AssertArrayResults.ReportResult(ExpectedsSize := DINT_TO_UDINT(SizeOfExpecteds),
                                ExpectedsTypeClass := IBaseLibrary.TypeClass.TYPE_ULINT,
                                ActualsSize := DINT_TO_UDINT(SizeOfActuals),
                                ActualsTypeClass := IBaseLibrary.TypeClass.TYPE_ULINT,
                                Message := Message,
                                TestInstancePath := TestInstancePath,
                                AlreadyReported => AlreadyReported);

IF NOT AlreadyReported AND NOT Equals THEN
    SetTestFailed(AssertionType := E_AssertionType.Type_Array_ULINT,
                  AssertionMessage := Message);

    IF NOT SizeEquals THEN
        Message := Tc2_Standard.CONCAT(STR1 := Message, STR2 := ', size of arrays not matching.');
        ExpectedString := 'SIZE = ';
        ExpectedString := Tc2_Standard.CONCAT(STR1 := ExpectedString, STR2 := DINT_TO_STRING(SizeOfExpecteds));
        ActualString := 'SIZE = ';
        ActualString := Tc2_Standard.CONCAT(STR1 := ActualString, STR2 := DINT_TO_STRING(SizeOfActuals));
    ELSE
        ExpectedString := 'ARRAY[';
        ExpectedString := Tc2_Standard.CONCAT(STR1 := ExpectedString, STR2 := DINT_TO_STRING(ExpectedsIndex));
        ExpectedString := Tc2_Standard.CONCAT(STR1 := ExpectedString, STR2 := '] = ');
        ExpectedString := Tc2_Standard.CONCAT(STR1 := ExpectedString, STR2 := ULINT_TO_STRING(Expecteds[ExpectedsIndex]));

        ActualString := 'ARRAY[';
        ActualString := Tc2_Standard.CONCAT(STR1 := ActualString, STR2 := DINT_TO_STRING(ActualsIndex));
        ActualString := Tc2_Standard.CONCAT(STR1 := ActualString, STR2 := '] = ');
        ActualString := Tc2_Standard.CONCAT(STR1 := ActualString, STR2 := ULINT_TO_STRING(Actuals[ActualsIndex]));
    END_IF

    AssertMessageFormatter.LogAssertFailure(Expected := ExpectedString,
                                            Actual := ActualString,
                                            Message := Message,
                                            TestInstancePath := TestInstancePath);
END_IF
END_METHOD

(*
    Asserts that two USINT arrays are equal. If they are not, an assertion error is created.
*)
METHOD PUBLIC AssertArrayEquals_USINT
VAR_IN_OUT
    Expecteds : ARRAY[*] OF USINT; // USINT array with expected values
    Actuals : ARRAY[*] OF USINT; // USINT array with actual values
END_VAR
VAR_INPUT
    Message : Tc2_System.T_MaxString; // The identifying message for the assertion error
END_VAR
VAR
    Equals : BOOL := TRUE;
    SizeEquals : BOOL := TRUE;
    Index : DINT;
    ExpectedString : Tc2_System.T_MaxString;
    ActualString : Tc2_System.T_MaxString;
    AlreadyReported : BOOL;
    TestInstancePath : Tc2_System.T_MaxString;
    SizeOfExpecteds : DINT;
    SizeOfActuals : DINT;
    ExpectedsIndex : DINT;
    ActualsIndex : DINT;
END_VAR
IF GVL_TcUnit.IgnoreCurrentTest OR GVL_TcUnit.CurrentTestIsFinished THEN
    RETURN;
END_IF

TestInstancePath := AddTestNameToInstancePath(FindTestSuiteInstancePath());

SizeOfExpecteds := ABS(UPPER_BOUND(Expecteds, 1) - LOWER_BOUND(Expecteds, 1)) + 1;
SizeOfActuals := ABS(UPPER_BOUND(Actuals, 1) - LOWER_BOUND(Actuals, 1)) + 1;

IF SizeOfExpecteds <> SizeOfActuals THEN
    Equals := FALSE;
    SizeEquals := FALSE;
ELSE
    (* Even though we know that both arrays are equal in size, the two arrays can start at two completely different
       indexes, which needs to be taken into account for. *)
    ExpectedsIndex := LOWER_BOUND(Expecteds, 1); // The start position for the expecteds
    ActualsIndex := LOWER_BOUND(Actuals, 1); // The start position for the actuals
    FOR Index := 1 TO SizeOfExpecteds BY 1 DO
        IF Expecteds[ExpectedsIndex] <> Actuals[ActualsIndex] THEN
            Equals := FALSE;
            EXIT;
        END_IF
        ExpectedsIndex := ExpectedsIndex + 1;
        ActualsIndex := ActualsIndex + 1;
    END_FOR
END_IF

AssertArrayResults.ReportResult(ExpectedsSize := DINT_TO_UDINT(SizeOfExpecteds),
                                ExpectedsTypeClass := IBaseLibrary.TypeClass.TYPE_USINT,
                                ActualsSize := DINT_TO_UDINT(SizeOfActuals),
                                ActualsTypeClass := IBaseLibrary.TypeClass.TYPE_USINT,
                                Message := Message,
                                TestInstancePath := TestInstancePath,
                                AlreadyReported => AlreadyReported);

IF NOT AlreadyReported AND NOT Equals THEN
    SetTestFailed(AssertionType := E_AssertionType.Type_Array_USINT,
                  AssertionMessage := Message);

    IF NOT SizeEquals THEN
        Message := Tc2_Standard.CONCAT(STR1 := Message, STR2 := ', size of arrays not matching.');
        ExpectedString := 'SIZE = ';
        ExpectedString := Tc2_Standard.CONCAT(STR1 := ExpectedString, STR2 := DINT_TO_STRING(SizeOfExpecteds));
        ActualString := 'SIZE = ';
        ActualString := Tc2_Standard.CONCAT(STR1 := ActualString, STR2 := DINT_TO_STRING(SizeOfActuals));
    ELSE
        ExpectedString := 'ARRAY[';
        ExpectedString := Tc2_Standard.CONCAT(STR1 := ExpectedString, STR2 := DINT_TO_STRING(ExpectedsIndex));
        ExpectedString := Tc2_Standard.CONCAT(STR1 := ExpectedString, STR2 := '] = ');
        ExpectedString := Tc2_Standard.CONCAT(STR1 := ExpectedString, STR2 := USINT_TO_STRING(Expecteds[ExpectedsIndex]));

        ActualString := 'ARRAY[';
        ActualString := Tc2_Standard.CONCAT(STR1 := ActualString, STR2 := DINT_TO_STRING(ActualsIndex));
        ActualString := Tc2_Standard.CONCAT(STR1 := ActualString, STR2 := '] = ');
        ActualString := Tc2_Standard.CONCAT(STR1 := ActualString, STR2 := USINT_TO_STRING(Actuals[ActualsIndex]));
    END_IF

    AssertMessageFormatter.LogAssertFailure(Expected := ExpectedString,
                                            Actual := ActualString,
                                            Message := Message,
                                            TestInstancePath := TestInstancePath);
END_IF
END_METHOD

(*
    Asserts that two WORD arrays are equal. If they are not, an assertion error is created.
*)
METHOD PUBLIC AssertArrayEquals_WORD
VAR_IN_OUT
    Expecteds : ARRAY[*] OF WORD; // WORD array with expected values
    Actuals : ARRAY[*] OF WORD; // WORD array with actual values
END_VAR
VAR_INPUT
    Message : Tc2_System.T_MaxString; // The identifying message for the assertion error
END_VAR
VAR
    Equals : BOOL := TRUE;
    SizeEquals : BOOL := TRUE;
    Index : DINT;
    ExpectedString : Tc2_System.T_MaxString;
    ActualString : Tc2_System.T_MaxString;
    AlreadyReported : BOOL;
    TestInstancePath : Tc2_System.T_MaxString;
    SizeOfExpecteds : DINT;
    SizeOfActuals : DINT;
    ExpectedDWordString : STRING;
    ActualDWordString : STRING;
    ExpectedsIndex : DINT;
    ActualsIndex : DINT;
END_VAR
IF GVL_TcUnit.IgnoreCurrentTest OR GVL_TcUnit.CurrentTestIsFinished THEN
    RETURN;
END_IF

TestInstancePath := AddTestNameToInstancePath(FindTestSuiteInstancePath());

SizeOfExpecteds := ABS(UPPER_BOUND(Expecteds, 1) - LOWER_BOUND(Expecteds, 1)) + 1;
SizeOfActuals := ABS(UPPER_BOUND(Actuals, 1) - LOWER_BOUND(Actuals, 1)) + 1;

IF SizeOfExpecteds <> SizeOfActuals THEN
    Equals := FALSE;
    SizeEquals := FALSE;
ELSE
    (* Even though we know that both arrays are equal in size, the two arrays can start at two completely different
       indexes, which needs to be taken into account for. *)
    ExpectedsIndex := LOWER_BOUND(Expecteds, 1); // The start position for the expecteds
    ActualsIndex := LOWER_BOUND(Actuals, 1); // The start position for the actuals
    FOR Index := 1 TO SizeOfExpecteds BY 1 DO
        IF Expecteds[ExpectedsIndex] <> Actuals[ActualsIndex] THEN
            Equals := FALSE;
            EXIT;
        END_IF
        ExpectedsIndex := ExpectedsIndex + 1;
        ActualsIndex := ActualsIndex + 1;
    END_FOR
END_IF

AssertArrayResults.ReportResult(ExpectedsSize := DINT_TO_UDINT(SizeOfExpecteds),
                                ExpectedsTypeClass := IBaseLibrary.TypeClass.TYPE_WORD,
                                ActualsSize := DINT_TO_UDINT(SizeOfActuals),
                                ActualsTypeClass := IBaseLibrary.TypeClass.TYPE_WORD,
                                Message := Message,
                                TestInstancePath := TestInstancePath,
                                AlreadyReported => AlreadyReported);

IF NOT AlreadyReported AND NOT Equals THEN
    SetTestFailed(AssertionType := E_AssertionType.Type_Array_WORD,
                  AssertionMessage := Message);

    IF NOT SizeEquals THEN
        Message := Tc2_System.CONCAT(STR1 := Message, STR2 := ', size of arrays not matching.');
        ExpectedString := 'SIZE = ';
        ExpectedString := Tc2_System.CONCAT(STR1 := ExpectedString, STR2 := DINT_TO_STRING(SizeOfExpecteds));
        ActualString := 'SIZE = ';
        ActualString := Tc2_System.CONCAT(STR1 := ActualString, STR2 := DINT_TO_STRING(SizeOfActuals));
    ELSE
        ExpectedDWordString := Tc2_Standard.CONCAT(STR1 := '0x',
                                                  STR2 := Tc2_Utilities.WORD_TO_HEXSTR(in := Expecteds[ExpectedsIndex],
                                                                                       iPrecision := 4,
                                                                                       bLoCase := FALSE));
        ExpectedString := 'ARRAY[';
        ExpectedString := Tc2_System.CONCAT(STR1 := ExpectedString, STR2 := DINT_TO_STRING(ExpectedsIndex));
        ExpectedString := Tc2_System.CONCAT(STR1 := ExpectedString, STR2 := '] = ');
        ExpectedString := Tc2_System.CONCAT(STR1 := ExpectedString, STR2 := ExpectedDWordString);

        ActualDWordString := Tc2_Standard.CONCAT(STR1 := '0x',
                                                 STR2 := Tc2_Utilities.WORD_TO_HEXSTR(in := Actuals[ActualsIndex],
                                                                                      iPrecision := 4,
                                                                                      bLoCase := FALSE));
        ActualString := 'ARRAY[';
        ActualString := Tc2_System.CONCAT(STR1 := ActualString, STR2 := DINT_TO_STRING(ActualsIndex));
        ActualString := Tc2_System.CONCAT(STR1 := ActualString, STR2 := '] = ');
        ActualString := Tc2_System.CONCAT(STR1 := ActualString, STR2 := ActualDWordString);
    END_IF

    AssertMessageFormatter.LogAssertFailure(Expected := ExpectedString,
                                            Actual := ActualString,
                                            Message := Message,
                                            TestInstancePath := TestInstancePath);
END_IF
END_METHOD

(*
    Asserts that two objects (of any type) are equal. If they are not, an assertion error is created.
    For REAL and LREAL it's recommended to use the AssertEquals_REAL or AssertEquals_LREAL respectively
    as these give the possibility to specify a delta between the expected and actual value.
*)
METHOD PUBLIC AssertEquals
VAR_INPUT
    Expected : ANY; // Expected value
    Actual : ANY; // The value to check against expected
    Message : Tc2_System.T_MaxString; // The identifying message for the assertion error
END_VAR
VAR
    Count : DINT;
    ExpectedDataString : Tc2_System.T_MaxString;
    ActualDataString : Tc2_System.T_MaxString;
    TestInstancePath : Tc2_System.T_MaxString;
    AlreadyReported : BOOL;

    boolExpected : BOOL;
    boolActual : BOOL;
    byteExpected : BYTE;
    byteActual : BYTE;
    dateExpected : DATE;
    dateActual : DATE;
    dateAndTimeExpected : DATE_AND_TIME;
    dateAndTimeActual : DATE_AND_TIME;
    dintExpected : DINT;
    dintActual : DINT;
    dwordExpected : DWORD;
    dwordActual : DWORD;
    intExpected : INT;
    intActual : INT;
    lintExpected : LINT;
    lintActual : LINT;
    lrealExpected : LREAL;
    lrealActual : LREAL;
    ltimeExpected : LTIME;
    ltimeActual : LTIME;
    lwordExpected : LWORD;
    lwordActual : LWORD;
    realExpected : REAL;
    realActual : REAL;
    sintExpected : SINT;
    sintActual : SINT;
    stringExpected : Tc2_System.T_MaxString;
    stringActual : Tc2_System.T_MaxString;
    wstringExpected : WSTRING(255);
    wstringActual : WSTRING(255);
    timeExpected : TIME;
    timeActual : TIME;
    timeOfDayExpected : TIME_OF_DAY;
    timeOfDayActual : TIME_OF_DAY;
    udintExpected : UDINT;
    udintActual : UDINT;
    uintExpected : UINT;
    uintActual : UINT;
    ulintExpected : ULINT;
    ulintActual : ULINT;
    usintExpected : USINT;
    usintActual : USINT;
    wordExpected : WORD;
    wordActual : WORD;

    (* ANY comparison variables *)
    DataTypesNotEquals : BOOL; // The data type of the two ANY input parameters are not equal
    DataSizeNotEquals : BOOL; // The data size of the two ANY input parameters are not equal
    DataContentNotEquals : BOOL; // The data content of the two ANY input parameters are not equal
    IteratorCounter : DINT;
END_VAR
IF GVL_TcUnit.IgnoreCurrentTest OR GVL_TcUnit.CurrentTestIsFinished THEN
    RETURN;
END_IF

(*
    This compares two instances of any object type and returns whether they
    are the same type, size and value or not. This is necessary for two reasons:
    1. So that we can know exactly what differs between the two input parameters
    2. It's not possible to do a comparison (= or <>) between two instances of ANY. 
*)
(* Check whether the type of the inputs differs *)
IF Expected.TypeClass <> Actual.TypeClass THEN
    DataTypesNotEquals := TRUE;
END_IF

(* Check whether the size of the inputs differs *)
IF NOT DataTypesNotEquals THEN
    (* Take special care of STRING and WSTRING, as these can be declared with different sizes,
       although their content might be the same *)
    IF UDINT_TO_INT(Expected.TypeClass) = IBaseLibrary.TypeClass.TYPE_STRING THEN
        Tc2_System.MEMCPY(destAddr := ADR(stringExpected), srcAddr := Expected.pValue, n := DINT_TO_UDINT(Expected.diSize));
        Tc2_System.MEMCPY(destAddr := ADR(stringActual), srcAddr := Actual.pValue, n := DINT_TO_UDINT(Actual.diSize));
        DataSizeNotEquals := Tc2_Standard.LEN(STR := stringExpected) <> Tc2_Standard.LEN(STR := stringActual);
    ELSIF UDINT_TO_INT(Expected.TypeClass) = IBaseLibrary.TypeClass.TYPE_WSTRING THEN
        Tc2_System.MEMCPY(destAddr := ADR(wstringExpected), srcAddr := Expected.pValue, n := DINT_TO_UDINT(Expected.diSize));
        Tc2_System.MEMCPY(destAddr := ADR(wstringActual), srcAddr := Actual.pValue, n := DINT_TO_UDINT(Actual.diSize));
        DataSizeNotEquals := Tc2_Standard.WLEN(STR := wstringExpected) <> Tc2_Standard.WLEN(STR := wstringActual);
    ELSIF (Expected.diSize <> Actual.diSize) THEN
        DataSizeNotEquals := TRUE;
    END_IF
END_IF

(* Even though the data type and size are equals, the contents may still differ *)
IF NOT DataTypesNotEquals AND NOT DataSizeNotEquals THEN
    // Compare each byte in the ANY-types
    FOR IteratorCounter := 0 TO Expected.diSize - 1 BY 1 DO
        IF Expected.pValue[IteratorCounter] <> Actual.pValue[IteratorCounter] THEN
            DataContentNotEquals := TRUE;
            EXIT;
        END_IF
    END_FOR
END_IF

(* First check whether the input data are any of the standard data types that are supported by TcUnit.
   In this case call the standard Assert-methods for that data. But before doing that we need to make sure
   that both the expected and actual:
   - Have both the same data type
   - Both have the same data size
*)
IF NOT DataTypesNotEquals AND NOT DataSizeNotEquals THEN

    (* BOOL *)
    IF UDINT_TO_INT(Expected.TypeClass) = IBaseLibrary.TypeClass.TYPE_BOOL THEN
        Tc2_System.MEMCPY(destAddr := ADR(boolExpected), srcAddr := Expected.pValue, n := SIZEOF(BOOL));
        Tc2_System.MEMCPY(destAddr := ADR(boolActual), srcAddr := Actual.pValue, n := SIZEOF(BOOL));
        AssertEquals_BOOL(Expected := boolExpected, Actual := boolActual, Message := Message);
        RETURN;
    END_IF

    (* BYTE *)
    IF UDINT_TO_INT(Expected.TypeClass) = IBaseLibrary.TypeClass.TYPE_BYTE THEN
        Tc2_System.MEMCPY(destAddr := ADR(byteExpected), srcAddr := Expected.pValue, n := SIZEOF(BYTE));
        Tc2_System.MEMCPY(destAddr := ADR(byteActual), srcAddr := Actual.pValue, n := SIZEOF(BYTE));
        AssertEquals_BYTE(Expected := byteExpected, Actual := byteActual, Message := Message);
        RETURN;
    END_IF

    (* DATE *)
    IF UDINT_TO_INT(Expected.TypeClass) = IBaseLibrary.TypeClass.TYPE_DATE THEN
        Tc2_System.MEMCPY(destAddr := ADR(dateExpected), srcAddr := Expected.pValue, n := SIZEOF(DATE));
        Tc2_System.MEMCPY(destAddr := ADR(dateActual), srcAddr := Actual.pValue, n := SIZEOF(DATE));
        AssertEquals_DATE(Expected := dateExpected, Actual := dateActual, Message := Message);
        RETURN;
    END_IF

    (* DATE_AND_TIME *)
    IF UDINT_TO_INT(Expected.TypeClass) = IBaseLibrary.TypeClass.TYPE_DATEANDTIME THEN
        Tc2_System.MEMCPY(destAddr := ADR(dateAndTimeExpected), srcAddr := Expected.pValue, n := SIZEOF(DATE_AND_TIME));
        Tc2_System.MEMCPY(destAddr := ADR(dateAndTimeActual), srcAddr := Actual.pValue, n := SIZEOF(DATE_AND_TIME));
        AssertEquals_DATE_AND_TIME(Expected := dateAndTimeExpected, Actual := dateAndTimeActual, Message := Message);
        RETURN;
    END_IF

    (* DINT *)
    IF UDINT_TO_INT(Expected.TypeClass) = IBaseLibrary.TypeClass.TYPE_DINT THEN
        Tc2_System.MEMCPY(destAddr := ADR(dintExpected), srcAddr := Expected.pValue, n := SIZEOF(DINT));
        Tc2_System.MEMCPY(destAddr := ADR(dintActual), srcAddr := Actual.pValue, n := SIZEOF(DINT));
        AssertEquals_DINT(Expected := dintExpected, Actual := dintActual, Message := Message);
        RETURN;
    END_IF

    (* DWORD *)
    IF UDINT_TO_INT(Expected.TypeClass) = IBaseLibrary.TypeClass.TYPE_DWORD THEN
        Tc2_System.MEMCPY(destAddr := ADR(dwordExpected), srcAddr := Expected.pValue, n := SIZEOF(DWORD));
        Tc2_System.MEMCPY(destAddr := ADR(dwordActual), srcAddr := Actual.pValue, n := SIZEOF(DWORD));
        AssertEquals_DWORD(Expected := dwordExpected, Actual := dwordActual, Message := Message);
        RETURN;
    END_IF

    (* INT *)
    IF UDINT_TO_INT(Expected.TypeClass) = IBaseLibrary.TypeClass.TYPE_INT THEN
        Tc2_System.MEMCPY(destAddr := ADR(intExpected), srcAddr := Expected.pValue, n := SIZEOF(INT));
        Tc2_System.MEMCPY(destAddr := ADR(intActual), srcAddr := Actual.pValue, n := SIZEOF(INT));
        AssertEquals_INT(Expected := intExpected, Actual := intActual, Message := Message);
        RETURN;
    END_IF

    (* LINT *)
    IF UDINT_TO_INT(Expected.TypeClass) = IBaseLibrary.TypeClass.TYPE_LINT THEN
        Tc2_System.MEMCPY(destAddr := ADR(lintExpected), srcAddr := Expected.pValue, n := SIZEOF(LINT));
        Tc2_System.MEMCPY(destAddr := ADR(lintActual), srcAddr := Actual.pValue, n := SIZEOF(LINT));
        AssertEquals_LINT(Expected := lintExpected, Actual := lintActual, Message := Message);
        RETURN;
    END_IF

    (* LREAL *)
    IF UDINT_TO_INT(Expected.TypeClass) = IBaseLibrary.TypeClass.TYPE_LREAL THEN
        Tc2_System.MEMCPY(destAddr := ADR(lrealExpected), srcAddr := Expected.pValue, n := SIZEOF(LREAL));
        Tc2_System.MEMCPY(destAddr := ADR(lrealActual), srcAddr := Actual.pValue, n := SIZEOF(LREAL));
        AssertEquals_LREAL(Expected := lrealExpected, Actual := lrealActual, Delta := 0.0, Message := Message);
        RETURN;
    END_IF

    (* LTIME *)
    IF UDINT_TO_INT(Expected.TypeClass) = IBaseLibrary.TypeClass.TYPE_LTIME THEN
        Tc2_System.MEMCPY(destAddr := ADR(ltimeExpected), srcAddr := Expected.pValue, n := SIZEOF(LTIME));
        Tc2_System.MEMCPY(destAddr := ADR(ltimeActual), srcAddr := Actual.pValue, n := SIZEOF(LTIME));
        AssertEquals_LTIME(Expected := ltimeExpected, Actual := ltimeActual, Message := Message);
        RETURN;
    END_IF

    (* LWORD *)
    IF UDINT_TO_INT(Expected.TypeClass) = IBaseLibrary.TypeClass.TYPE_LWORD THEN
        Tc2_System.MEMCPY(destAddr := ADR(lwordExpected), srcAddr := Expected.pValue, n := SIZEOF(LWORD));
        Tc2_System.MEMCPY(destAddr := ADR(lwordActual), srcAddr := Actual.pValue, n := SIZEOF(LWORD));
        AssertEquals_LWORD(Expected := lwordExpected, Actual := lwordActual, Message := Message);
        RETURN;
    END_IF

    (* REAL *)
    IF UDINT_TO_INT(Expected.TypeClass) = IBaseLibrary.TypeClass.TYPE_REAL THEN
        Tc2_System.MEMCPY(destAddr := ADR(realExpected), srcAddr := Expected.pValue, n := SIZEOF(REAL));
        Tc2_System.MEMCPY(destAddr := ADR(realActual), srcAddr := Actual.pValue, n := SIZEOF(REAL));
        AssertEquals_REAL(Expected := realExpected, Actual := realActual, Delta := 0.0, Message := Message);
        RETURN;
    END_IF

    (* SINT *)
    IF UDINT_TO_INT(Expected.TypeClass) = IBaseLibrary.TypeClass.TYPE_SINT THEN
        Tc2_System.MEMCPY(destAddr := ADR(sintExpected), srcAddr := Expected.pValue, n := SIZEOF(SINT));
        Tc2_System.MEMCPY(destAddr := ADR(sintActual), srcAddr := Actual.pValue, n := SIZEOF(SINT));
        AssertEquals_SINT(Expected := sintExpected, Actual := sintActual, Message := Message);
        RETURN;
    END_IF

    (* STRING *)
    IF UDINT_TO_INT(Expected.TypeClass) = IBaseLibrary.TypeClass.TYPE_STRING THEN
        Tc2_System.MEMCPY(destAddr := ADR(stringExpected), srcAddr := Expected.pValue, n := DINT_TO_UDINT(Expected.diSize));
        Tc2_System.MEMCPY(destAddr := ADR(stringActual), srcAddr := Actual.pValue, n := DINT_TO_UDINT(Actual.diSize));
        AssertEquals_STRING(Expected := stringExpected, Actual := stringActual, Message := Message);
        RETURN;
    END_IF

    (* WSTRING *)
    IF UDINT_TO_INT(Expected.TypeClass) = IBaseLibrary.TypeClass.TYPE_WSTRING THEN
        Tc2_System.MEMCPY(destAddr := ADR(wstringExpected), srcAddr := Expected.pValue, n := DINT_TO_UDINT(Expected.diSize));
        Tc2_System.MEMCPY(destAddr := ADR(wstringActual), srcAddr := Actual.pValue, n := DINT_TO_UDINT(Actual.diSize));
        AssertEquals_WSTRING(Expected := wstringExpected, Actual := wstringActual, Message := Message);
        RETURN;
    END_IF

    (* TIME *)
    IF UDINT_TO_INT(Expected.TypeClass) = IBaseLibrary.TypeClass.TYPE_TIME THEN
        Tc2_System.MEMCPY(destAddr := ADR(timeExpected), srcAddr := Expected.pValue, n := SIZEOF(TIME));
        Tc2_System.MEMCPY(destAddr := ADR(timeActual), srcAddr := Actual.pValue, n := SIZEOF(TIME));
        AssertEquals_TIME(Expected := timeExpected, Actual := timeActual, Message := Message);
        RETURN;
    END_IF

    (* TIME_OF_DAY *)
    IF UDINT_TO_INT(Expected.TypeClass) = IBaseLibrary.TypeClass.TYPE_TIMEOFDAY THEN
        Tc2_System.MEMCPY(destAddr := ADR(timeOfDayExpected), srcAddr := Expected.pValue, n := SIZEOF(TIME_OF_DAY));
        Tc2_System.MEMCPY(destAddr := ADR(timeOfDayActual), srcAddr := Actual.pValue, n := SIZEOF(TIME_OF_DAY));
        AssertEquals_TIME_OF_DAY(Expected := timeOfDayExpected, Actual := timeOfDayActual, Message := Message);
        RETURN;
    END_IF

    (* UDINT *)
    IF UDINT_TO_INT(Expected.TypeClass) = IBaseLibrary.TypeClass.TYPE_UDINT THEN
        Tc2_System.MEMCPY(destAddr := ADR(udintExpected), srcAddr := Expected.pValue, n := SIZEOF(UDINT));
        Tc2_System.MEMCPY(destAddr := ADR(udintActual), srcAddr := Actual.pValue, n := SIZEOF(UDINT));
        AssertEquals_UDINT(Expected := udintExpected, Actual := udintActual, Message := Message);
        RETURN;
    END_IF

    (* UINT *)
    IF UDINT_TO_INT(Expected.TypeClass) = IBaseLibrary.TypeClass.TYPE_UINT THEN
        Tc2_System.MEMCPY(destAddr := ADR(uintExpected), srcAddr := Expected.pValue, n := SIZEOF(UINT));
        Tc2_System.MEMCPY(destAddr := ADR(uintActual), srcAddr := Actual.pValue, n := SIZEOF(UINT));
        AssertEquals_UINT(Expected := uintExpected, Actual := uintActual, Message := Message);
        RETURN;
    END_IF

    (* ULINT *)
    IF UDINT_TO_INT(Expected.TypeClass) = IBaseLibrary.TypeClass.TYPE_ULINT THEN
        Tc2_System.MEMCPY(destAddr := ADR(ulintExpected), srcAddr := Expected.pValue, n := SIZEOF(ULINT));
        Tc2_System.MEMCPY(destAddr := ADR(ulintActual), srcAddr := Actual.pValue, n := SIZEOF(ULINT));
        AssertEquals_ULINT(Expected := ulintExpected, Actual := ulintActual, Message := Message);
        RETURN;
    END_IF

    (* USINT *)
    IF UDINT_TO_INT(Expected.TypeClass) = IBaseLibrary.TypeClass.TYPE_USINT THEN
        Tc2_System.MEMCPY(destAddr := ADR(usintExpected), srcAddr := Expected.pValue, n := SIZEOF(USINT));
        Tc2_System.MEMCPY(destAddr := ADR(usintActual), srcAddr := Actual.pValue, n := SIZEOF(USINT));
        AssertEquals_USINT(Expected := usintExpected, Actual := usintActual, Message := Message);
        RETURN;
    END_IF

    (* WORD *)
    IF UDINT_TO_INT(Expected.TypeClass) = IBaseLibrary.TypeClass.TYPE_WORD THEN
        Tc2_System.MEMCPY(destAddr := ADR(wordExpected), srcAddr := Expected.pValue, n := SIZEOF(WORD));
        Tc2_System.MEMCPY(destAddr := ADR(wordActual), srcAddr := Actual.pValue, n := SIZEOF(WORD));
        AssertEquals_WORD(Expected := wordExpected, Actual := wordActual, Message := Message);
        RETURN;
    END_IF

END_IF

(* If we've come to this row, it means that the data input is not any of the standard primitive data types, and thus
   we need to do special handling *)
TestInstancePath := AddTestNameToInstancePath(TestInstancePath := FindTestSuiteInstancePath());

IF DataTypesNotEquals THEN
    ExpectedDataString := Tc2_Standard.CONCAT(STR1 := '(Type class = ', STR2 := F_AnyTypeClassToString((Expected.TypeClass)));
    ExpectedDataString := Tc2_Standard.CONCAT(STR1 := ExpectedDataString, STR2 := ')');
    ActualDataString := Tc2_Standard.CONCAT(STR1 := '(Type class = ', STR2 := F_AnyTypeClassToString(Actual.TypeClass));
    ActualDataString := Tc2_Standard.CONCAT(STR1 := ActualDataString, STR2 := ')');
ELSIF DataSizeNotEquals THEN
    (* Take special care of STRING and WSTRING, as these can be declared with different sizes,
       although their content might be the same *)
    IF UDINT_TO_INT(Expected.TypeClass) = IBaseLibrary.TypeClass.TYPE_STRING THEN
        Tc2_System.MEMCPY(destAddr := ADR(stringExpected), srcAddr := Expected.pValue, n := DINT_TO_UDINT(Expected.diSize));
        Tc2_System.MEMCPY(destAddr := ADR(stringActual), srcAddr := Actual.pValue, n := DINT_TO_UDINT(Actual.diSize));
        ExpectedDataString := Tc2_Standard.CONCAT(STR1 := '(Data size (LEN) = ', STR2 := INT_TO_STRING(Tc2_Standard.LEN(STR := stringExpected)));
        ActualDataString := Tc2_Standard.CONCAT(STR1 := '(Data size (LEN) = ', STR2 := INT_TO_STRING(Tc2_Standard.LEN(STR := stringActual)));
    ELSIF UDINT_TO_INT(Expected.TypeClass) = IBaseLibrary.TypeClass.TYPE_WSTRING THEN
        Tc2_System.MEMCPY(destAddr := ADR(wstringExpected), srcAddr := Expected.pValue, n := DINT_TO_UDINT(Expected.diSize));
        Tc2_System.MEMCPY(destAddr := ADR(wstringActual), srcAddr := Actual.pValue, n := DINT_TO_UDINT(Actual.diSize));
        ExpectedDataString := Tc2_Standard.CONCAT(STR1 := '(Data size (WLEN) = ', STR2 := INT_TO_STRING(Tc2_Standard.WLEN(STR := wstringExpected)));
        ActualDataString := Tc2_Standard.CONCAT(STR1 := '(Data size (WLEN) = ', STR2 := INT_TO_STRING(Tc2_Standard.WLEN(STR := wstringActual)));
    ELSE
        ExpectedDataString := Tc2_Standard.CONCAT(STR1 := '(Data size = ', STR2 := DINT_TO_STRING(Expected.diSize));
        ActualDataString := Tc2_Standard.CONCAT(STR1 := '(Data size = ', STR2 := DINT_TO_STRING(Actual.diSize));
    END_IF
    ExpectedDataString := Tc2_Standard.CONCAT(STR1 := ExpectedDataString, STR2 := ')');
    ActualDataString := Tc2_Standard.CONCAT(STR1 := ActualDataString, STR2 := ')');
ELSIF DataContentNotEquals THEN
    FOR Count := 0 TO MIN(Expected.diSize-1, 38) BY 1 DO // One byte will equal two characters (example: 255 = 0xff, 1 = 0x01)
        ExpectedDataString := Tc2_Standard.CONCAT(STR1 := ExpectedDataString,
                                                  STR2 := Tc2_Utilities.BYTE_TO_HEXSTR(in := Expected.pValue[Count],
                                                                                       iPrecision := 2,
                                                                                       bLoCase := FALSE));
    END_FOR
    ExpectedDataString := Tc2_Standard.CONCAT(STR1 := '0x', STR2 := ExpectedDataString);

    FOR Count := 0 TO MIN(Actual.diSize-1, 38) BY 1 DO // One byte will equal two characters (example: 255 = 0xff, 1 = 0x01)
        ActualDataString := Tc2_Standard.CONCAT(STR1 := ActualDataString,
                                                STR2 := Tc2_Utilities.BYTE_TO_HEXSTR(in := Actual.pValue[Count],
                                                                                     iPrecision := 2,
                                                                                     bLoCase := FALSE));
    END_FOR
    ActualDataString := Tc2_Standard.CONCAT(STR1 := '0x', STR2 := ActualDataString);
END_IF

AssertResults.ReportResult(ExpectedSize := DINT_TO_UDINT(Expected.diSize),
                           ExpectedTypeClass := UDINT_TO_INT(Expected.TypeClass),
                           ExpectedValue := Expected.pValue,
                           ActualSize := DINT_TO_UDINT(Actual.diSize),
                           ActualTypeClass := UDINT_TO_INT(Actual.TypeClass),
                           ActualValue := Actual.pValue,
                           Message := Message,
                           TestInstancePath := TestInstancePath,
                           AlreadyReported => AlreadyReported);

IF NOT AlreadyReported AND (DataTypesNotEquals OR DataSizeNotEquals OR DataContentNotEquals) THEN
    SetTestFailed(AssertionType := E_AssertionType.Type_ANY,
                  AssertionMessage := Message);

    AssertMessageFormatter.LogAssertFailure(Expected := ExpectedDataString,
                                            Actual := ActualDataString,
                                            Message := Message,
                                            TestInstancePath := TestInstancePath);
END_IF
END_METHOD

(*
    Asserts that two BOOLs are equal. If they are not, an assertion error is created.
*)
METHOD PUBLIC AssertEquals_BOOL
VAR_INPUT
    Expected : BOOL; // BOOL expected value
    Actual : BOOL; // BOOL actual value
    Message : Tc2_System.T_MaxString; // The identifying message for the assertion error
END_VAR
VAR
    AlreadyReported : BOOL;
    TestInstancePath : Tc2_System.T_MaxString;
END_VAR
IF GVL_TcUnit.IgnoreCurrentTest OR GVL_TcUnit.CurrentTestIsFinished THEN
    RETURN;
END_IF

TestInstancePath := AddTestNameToInstancePath(TestInstancePath := FindTestSuiteInstancePath());

AssertResults.ReportResult(ExpectedSize := SIZEOF(Expected),
                           ExpectedTypeClass := IBaseLibrary.TypeClass.TYPE_BOOL,
                           ExpectedValue := ADR(Expected),
                           ActualSize := SIZEOF(Actual),
                           ActualTypeClass := IBaseLibrary.TypeClass.TYPE_BOOL,
                           ActualValue := ADR(Actual),
                           Message := Message,
                           TestInstancePath := TestInstancePath,
                           AlreadyReported => AlreadyReported);

IF NOT AlreadyReported AND Expected <> Actual THEN
    SetTestFailed(AssertionType := E_AssertionType.Type_BOOL,
                  AssertionMessage := Message);

    AssertMessageFormatter.LogAssertFailure(Expected := BOOL_TO_STRING(Expected),
                                            Actual := BOOL_TO_STRING(Actual),
                                            Message := Message,
                                            TestInstancePath := TestInstancePath);
END_IF
END_METHOD

(*
    Asserts that two BYTEs are equal. If they are not, an assertion error is created.
*)
METHOD PUBLIC AssertEquals_BYTE
VAR_INPUT
    Expected : BYTE; // BYTE expected value
    Actual : BYTE; // BYTE actual value
    Message : Tc2_System.T_MaxString; // The identifying message for the assertion error
END_VAR
VAR
    TestInstancePath : Tc2_System.T_MaxString;
    AlreadyReported : BOOL;
END_VAR
IF GVL_TcUnit.IgnoreCurrentTest OR GVL_TcUnit.CurrentTestIsFinished THEN
    RETURN;
END_IF

TestInstancePath := AddTestNameToInstancePath(TestInstancePath := FindTestSuiteInstancePath());

AssertResults.ReportResult(ExpectedSize := SIZEOF(Expected),
                           ExpectedTypeClass := IBaseLibrary.TypeClass.TYPE_BYTE,
                           ExpectedValue := ADR(Expected),
                           ActualSize := SIZEOF(Actual),
                           ActualTypeClass := IBaseLibrary.TypeClass.TYPE_BYTE,
                           ActualValue := ADR(Actual),
                           Message := Message,
                           TestInstancePath := TestInstancePath,
                           AlreadyReported => AlreadyReported);

IF NOT AlreadyReported AND Expected <> Actual THEN
    SetTestFailed(AssertionType := E_AssertionType.Type_BYTE,
                  AssertionMessage := Message);

    AssertMessageFormatter.LogAssertFailure(Expected := Tc2_Standard.CONCAT(
                                                       STR1 := '0x',
                                                       STR2 := Tc2_Utilities.BYTE_TO_HEXSTR(in := Expected,
                                                                                            iPrecision := 2,
                                                                                            bLoCase := FALSE)),
                                            Actual := Tc2_Standard.CONCAT(
                                                       STR1 := '0x',
                                                       STR2 := Tc2_Utilities.BYTE_TO_HEXSTR(in := Actual,
                                                                                            iPrecision := 2,
                                                                                            bLoCase := FALSE)),
                                            Message := Message,
                                            TestInstancePath := TestInstancePath);
END_IF
END_METHOD

(*
    Asserts that two DATEs are equal. If they are not, an assertion error is created.
*)
METHOD PUBLIC AssertEquals_DATE
VAR_INPUT
    Expected : DATE; // DATE expected value
    Actual : DATE; // DATE actual value
    Message : Tc2_System.T_MaxString; // The identifying message for the assertion error
END_VAR
VAR
    TestInstancePath : Tc2_System.T_MaxString;
    AlreadyReported : BOOL;
END_VAR
IF GVL_TcUnit.IgnoreCurrentTest OR GVL_TcUnit.CurrentTestIsFinished THEN
    RETURN;
END_IF

TestInstancePath := AddTestNameToInstancePath(TestInstancePath := FindTestSuiteInstancePath());

AssertResults.ReportResult(ExpectedSize := SIZEOF(Expected),
                           ExpectedTypeClass := IBaseLibrary.TypeClass.TYPE_DATE,
                           ExpectedValue := ADR(Expected),
                           ActualSize := SIZEOF(Actual),
                           ActualTypeClass := IBaseLibrary.TypeClass.TYPE_DATE,
                           ActualValue := ADR(Actual),
                           Message := Message,
                           TestInstancePath := TestInstancePath,
                           AlreadyReported => AlreadyReported);

IF NOT AlreadyReported AND Expected <> Actual THEN
    SetTestFailed(AssertionType := E_AssertionType.Type_DATE,
                  AssertionMessage := Message);

    AssertMessageFormatter.LogAssertFailure(Expected := DATE_TO_STRING(Expected),
                                            Actual := DATE_TO_STRING(Actual),
                                            Message := Message,
                                            TestInstancePath := TestInstancePath);
END_IF
END_METHOD

(*
    Asserts that two DATE_AND_TIMEs are equal. If they are not, an assertion error is created.
*)
METHOD PUBLIC AssertEquals_DATE_AND_TIME
VAR_INPUT
    Expected : DATE_AND_TIME; // DATE_AND_TIME expected value
    Actual : DATE_AND_TIME; // DATE_AND_TIME actual value
    Message : Tc2_System.T_MaxString; // The identifying message for the assertion error
END_VAR
VAR
    TestInstancePath : Tc2_System.T_MaxString;
    AlreadyReported : BOOL;
END_VAR
IF GVL_TcUnit.IgnoreCurrentTest OR GVL_TcUnit.CurrentTestIsFinished THEN
    RETURN;
END_IF

TestInstancePath := AddTestNameToInstancePath(TestInstancePath := FindTestSuiteInstancePath());

AssertResults.ReportResult(ExpectedSize := SIZEOF(Expected),
                           ExpectedTypeClass := IBaseLibrary.TypeClass.TYPE_DATEANDTIME,
                           ExpectedValue := ADR(Expected),
                           ActualSize := SIZEOF(Actual),
                           ActualTypeClass := IBaseLibrary.TypeClass.TYPE_DATEANDTIME,
                           ActualValue := ADR(Actual),
                           Message := Message,
                           TestInstancePath := TestInstancePath,
                           AlreadyReported => AlreadyReported);

IF NOT AlreadyReported AND Expected <> Actual THEN
    SetTestFailed(AssertionType := E_AssertionType.Type_DATE_AND_TIME,
                  AssertionMessage := Message);

    AssertMessageFormatter.LogAssertFailure(Expected := DT_TO_STRING(Expected),
                                            Actual := DT_TO_STRING(Actual),
                                            Message := Message,
                                            TestInstancePath := TestInstancePath);
END_IF
END_METHOD

(*
    Asserts that two DINTs are equal. If they are not, an assertion error is created.
*)
METHOD PUBLIC AssertEquals_DINT
VAR_INPUT
    Expected : DINT; // DINT expected value
    Actual : DINT; // DINT actual value
    Message : Tc2_System.T_MaxString; // The identifying message for the assertion error
END_VAR
VAR
    TestInstancePath : Tc2_System.T_MaxString;
    AlreadyReported : BOOL;
END_VAR
IF GVL_TcUnit.IgnoreCurrentTest OR GVL_TcUnit.CurrentTestIsFinished THEN
    RETURN;
END_IF

TestInstancePath := AddTestNameToInstancePath(TestInstancePath := FindTestSuiteInstancePath());

AssertResults.ReportResult(ExpectedSize := SIZEOF(Expected),
                           ExpectedTypeClass := IBaseLibrary.TypeClass.TYPE_DINT,
                           ExpectedValue := ADR(Expected),
                           ActualSize := SIZEOF(Actual),
                           ActualTypeClass := IBaseLibrary.TypeClass.TYPE_DINT,
                           ActualValue := ADR(Actual),
                           Message := Message,
                           TestInstancePath := TestInstancePath,
                           AlreadyReported => AlreadyReported);

IF NOT AlreadyReported AND Expected <> Actual THEN
    SetTestFailed(AssertionType := E_AssertionType.Type_DINT,
                  AssertionMessage := Message);

    AssertMessageFormatter.LogAssertFailure(Expected := DINT_TO_STRING(Expected),
                                            Actual := DINT_TO_STRING(Actual),
                                            Message := Message,
                                            TestInstancePath := TestInstancePath);
END_IF
END_METHOD

(*
    Asserts that two DWORDs are equal. If they are not, an assertion error is created.
*)
METHOD PUBLIC AssertEquals_DWORD
VAR_INPUT
    Expected : DWORD; // DWORD expected value
    Actual : DWORD; // DWORD actual value
    Message : Tc2_System.T_MaxString; // The identifying message for the assertion error
END_VAR
VAR
    TestInstancePath : Tc2_System.T_MaxString;
    AlreadyReported : BOOL;
END_VAR
IF GVL_TcUnit.IgnoreCurrentTest OR GVL_TcUnit.CurrentTestIsFinished THEN
    RETURN;
END_IF

TestInstancePath := AddTestNameToInstancePath(TestInstancePath := FindTestSuiteInstancePath());

AssertResults.ReportResult(ExpectedSize := SIZEOF(Expected),
                           ExpectedTypeClass := IBaseLibrary.TypeClass.TYPE_DWORD,
                           ExpectedValue := ADR(Expected),
                           ActualSize := SIZEOF(Actual),
                           ActualTypeClass := IBaseLibrary.TypeClass.TYPE_DWORD,
                           ActualValue := ADR(Actual),
                           Message := Message,
                           TestInstancePath := TestInstancePath,
                           AlreadyReported => AlreadyReported);

IF NOT AlreadyReported AND Expected <> Actual THEN
    SetTestFailed(AssertionType := E_AssertionType.Type_DWORD,
                  AssertionMessage := Message);

    AssertMessageFormatter.LogAssertFailure(Expected := Tc2_Standard.CONCAT(
                                                            STR1 := '0x',
                                                            STR2 := Tc2_Utilities.DWORD_TO_HEXSTR(in := Expected,
                                                                                                  iPrecision := 8,
                                                                                                  bLoCase := FALSE)),
                                            Actual := Tc2_Standard.CONCAT(
                                                           STR1 := '0x',
                                                           STR2 := Tc2_Utilities.DWORD_TO_HEXSTR(in := Actual,
                                                                                                 iPrecision := 8,
                                                                                                 bLoCase := FALSE)),
                                            Message := Message,
                                            TestInstancePath := TestInstancePath);
END_IF
END_METHOD

(*
    Asserts that two INTs are equal. If they are not, an assertion error is created.
*)
METHOD PUBLIC AssertEquals_INT
VAR_INPUT
    Expected : INT; // INT expected value
    Actual : INT; // INT actual value
    Message : Tc2_System.T_MaxString; // The identifying message for the assertion error
END_VAR
VAR
    TestInstancePath : Tc2_System.T_MaxString;
    AlreadyReported : BOOL;
END_VAR
IF GVL_TcUnit.IgnoreCurrentTest OR GVL_TcUnit.CurrentTestIsFinished THEN
    RETURN;
END_IF

TestInstancePath := AddTestNameToInstancePath(TestInstancePath := FindTestSuiteInstancePath());

AssertResults.ReportResult(ExpectedSize := SIZEOF(Expected),
                           ExpectedTypeClass := IBaseLibrary.TypeClass.TYPE_INT,
                           ExpectedValue := ADR(Expected),
                           ActualSize := SIZEOF(Actual),
                           ActualTypeClass := IBaseLibrary.TypeClass.TYPE_INT,
                           ActualValue := ADR(Actual),
                           Message := Message,
                           TestInstancePath := TestInstancePath,
                           AlreadyReported => AlreadyReported);

IF NOT AlreadyReported AND Expected <> Actual THEN
    SetTestFailed(AssertionType := E_AssertionType.Type_INT,
                  AssertionMessage := Message);

    AssertMessageFormatter.LogAssertFailure(Expected := INT_TO_STRING(Expected),
                                            Actual := INT_TO_STRING(Actual),
                                            Message := Message,
                                            TestInstancePath := TestInstancePath);
END_IF
END_METHOD

(*
    Asserts that two LINTs are equal. If they are not, an assertion error is created.
*)
METHOD PUBLIC AssertEquals_LINT
VAR_INPUT
    Expected : LINT; // LINT expected value
    Actual : LINT; // LINT actual value
    Message : Tc2_System.T_MaxString; // The identifying message for the assertion error
END_VAR
VAR
    TestInstancePath : Tc2_System.T_MaxString;
    AlreadyReported : BOOL;
END_VAR
IF GVL_TcUnit.IgnoreCurrentTest OR GVL_TcUnit.CurrentTestIsFinished THEN
    RETURN;
END_IF

TestInstancePath := AddTestNameToInstancePath(TestInstancePath := FindTestSuiteInstancePath());

AssertResults.ReportResult(ExpectedSize := SIZEOF(Expected),
                           ExpectedTypeClass := IBaseLibrary.TypeClass.TYPE_LINT,
                           ExpectedValue := ADR(Expected),
                           ActualSize := SIZEOF(Actual),
                           ActualTypeClass := IBaseLibrary.TypeClass.TYPE_LINT,
                           ActualValue := ADR(Actual),
                           Message := Message,
                           TestInstancePath := TestInstancePath,
                           AlreadyReported => AlreadyReported);

IF NOT AlreadyReported AND Expected <> Actual THEN
    SetTestFailed(AssertionType := E_AssertionType.Type_LINT,
                  AssertionMessage := Message);

    AssertMessageFormatter.LogAssertFailure(Expected := LINT_TO_STRING(Expected),
                                            Actual := LINT_TO_STRING(Actual),
                                            Message := Message,
                                            TestInstancePath := TestInstancePath);
END_IF
END_METHOD

(*
    Asserts that two LREALs are equal to within a positive delta. If they are not, an assertion error is created.
*)
METHOD PUBLIC AssertEquals_LREAL
VAR_INPUT
    Expected : LREAL; // LREAL expected value
    Actual : LREAL; // LREAL actual value
    Delta : LREAL; // The maximum delta between the absolute value of expected and actual for which both numbers are still considered equal
    Message : Tc2_System.T_MaxString; // The identifying message for the assertion error
END_VAR
VAR
    TestInstancePath : Tc2_System.T_MaxString;
    AlreadyReported : BOOL;
END_VAR
IF GVL_TcUnit.IgnoreCurrentTest OR GVL_TcUnit.CurrentTestIsFinished THEN
    RETURN;
END_IF

TestInstancePath := AddTestNameToInstancePath(TestInstancePath := FindTestSuiteInstancePath());

AssertResults.ReportResult(ExpectedSize := SIZEOF(Expected),
                           ExpectedTypeClass := IBaseLibrary.TypeClass.TYPE_LREAL,
                           ExpectedValue := ADR(Expected),
                           ActualSize := SIZEOF(Actual),
                           ActualTypeClass := IBaseLibrary.TypeClass.TYPE_LREAL,
                           ActualValue := ADR(Actual),
                           Message := Message,
                           TestInstancePath := TestInstancePath,
                           AlreadyReported => AlreadyReported);

IF NOT AlreadyReported AND ABS(Expected - Actual) > Delta THEN
    SetTestFailed(AssertionType := E_AssertionType.Type_LREAL,
                  AssertionMessage := Message);

    AssertMessageFormatter.LogAssertFailure(Expected := LREAL_TO_STRING(Expected),
                                            Actual := LREAL_TO_STRING(Actual),
                                            Message := Message,
                                            TestInstancePath := TestInstancePath);
END_IF
END_METHOD

(*
    Asserts that two LTIMEs are equal. If they are not, an assertion error is created.
*)
METHOD PUBLIC AssertEquals_LTIME
VAR_INPUT
    Expected : LTIME; // LTIME expected value
    Actual : LTIME; // LTIME actual value
    Message : Tc2_System.T_MaxString; // The identifying message for the assertion error
END_VAR
VAR
    TestInstancePath : Tc2_System.T_MaxString;
    AlreadyReported : BOOL;
END_VAR
IF GVL_TcUnit.IgnoreCurrentTest OR GVL_TcUnit.CurrentTestIsFinished THEN
    RETURN;
END_IF

TestInstancePath := AddTestNameToInstancePath(TestInstancePath := FindTestSuiteInstancePath());

AssertResults.ReportResult(ExpectedSize := SIZEOF(Expected),
                           ExpectedTypeClass := IBaseLibrary.TypeClass.TYPE_LTIME,
                           ExpectedValue := ADR(Expected),
                           ActualSize := SIZEOF(Actual),
                           ActualTypeClass := IBaseLibrary.TypeClass.TYPE_LTIME,
                           ActualValue := ADR(Actual),
                           Message := Message,
                           TestInstancePath := TestInstancePath,
                           AlreadyReported => AlreadyReported);

IF NOT AlreadyReported AND Expected <> Actual THEN
    SetTestFailed(AssertionType := E_AssertionType.Type_LTIME,
                  AssertionMessage := Message);

    AssertMessageFormatter.LogAssertFailure(Expected := LTIME_TO_STRING(Expected),
                                            Actual := LTIME_TO_STRING(Actual),
                                            Message := Message,
                                            TestInstancePath := TestInstancePath);
END_IF
END_METHOD

(*
    Asserts that two LWORDs are equal. If they are not, an assertion error is created.
*)
METHOD PUBLIC AssertEquals_LWORD
VAR_INPUT
    Expected : LWORD; // LWORD expected value
    Actual : LWORD; // LWORD actual value
    Message : Tc2_System.T_MaxString; // The identifying message for the assertion error
END_VAR
VAR
    TestInstancePath : Tc2_System.T_MaxString;
    AlreadyReported : BOOL;
END_VAR
IF GVL_TcUnit.IgnoreCurrentTest OR GVL_TcUnit.CurrentTestIsFinished THEN
    RETURN;
END_IF

TestInstancePath := AddTestNameToInstancePath(TestInstancePath := FindTestSuiteInstancePath());

AssertResults.ReportResult(ExpectedSize := SIZEOF(Expected),
                           ExpectedTypeClass := IBaseLibrary.TypeClass.TYPE_LWORD,
                           ExpectedValue := ADR(Expected),
                           ActualSize := SIZEOF(Actual),
                           ActualTypeClass := IBaseLibrary.TypeClass.TYPE_LWORD,
                           ActualValue := ADR(Actual),
                           Message := Message,
                           TestInstancePath := TestInstancePath,
                           AlreadyReported => AlreadyReported);

IF NOT AlreadyReported AND Expected <> Actual THEN
    SetTestFailed(AssertionType := E_AssertionType.Type_LWORD,
                  AssertionMessage := Message);

    AssertMessageFormatter.LogAssertFailure(Expected := Tc2_Standard.CONCAT(
                                                            STR1 := '0x',
                                                            STR2 := Tc2_Utilities.LWORD_TO_HEXSTR(in := Expected,
                                                                                                  iPrecision := 16,
                                                                                                  bLoCase := FALSE)),
                                            Actual := Tc2_Standard.CONCAT(
                                                            STR1 := '0x',
                                                            STR2 := Tc2_Utilities.LWORD_TO_HEXSTR(in := Actual,
                                                                                                  iPrecision := 16,
                                                                                                  bLoCase := FALSE)),
                                            Message := Message,
                                            TestInstancePath := TestInstancePath);
END_IF
END_METHOD

(*
    Asserts that two REALs are equal to within a positive delta. If they are not, an assertion error is created.
*)
METHOD PUBLIC AssertEquals_REAL
VAR_INPUT
    Expected : REAL; // REAL expected value
    Actual : REAL; // REAL actual value
    Delta : REAL;  // The maximum delta between the absolute value of expected and actual for which both numbers are still considered equal
    Message : Tc2_System.T_MaxString; // The identifying message for the assertion error
END_VAR
VAR
    TestInstancePath : Tc2_System.T_MaxString;
    AlreadyReported : BOOL;
END_VAR
IF GVL_TcUnit.IgnoreCurrentTest OR GVL_TcUnit.CurrentTestIsFinished THEN
    RETURN;
END_IF

TestInstancePath := AddTestNameToInstancePath(TestInstancePath := FindTestSuiteInstancePath());

AssertResults.ReportResult(ExpectedSize := SIZEOF(Expected),
                           ExpectedTypeClass := IBaseLibrary.TypeClass.TYPE_REAL,
                           ExpectedValue := ADR(Expected),
                           ActualSize := SIZEOF(Actual),
                           ActualTypeClass := IBaseLibrary.TypeClass.TYPE_REAL,
                           ActualValue := ADR(Actual),
                           Message := Message,
                           TestInstancePath := TestInstancePath,
                           AlreadyReported => AlreadyReported);

IF NOT AlreadyReported AND ABS(Expected - Actual) > Delta THEN
    SetTestFailed(AssertionType := E_AssertionType.Type_REAL,
                  AssertionMessage := Message);

    AssertMessageFormatter.LogAssertFailure(Expected := REAL_TO_STRING(Expected),
                                            Actual := REAL_TO_STRING(Actual),
                                            Message := Message,
                                            TestInstancePath := TestInstancePath);
END_IF
END_METHOD

(*
    Asserts that two SINTs are equal. If they are not, an assertion error is created.
*)
METHOD PUBLIC AssertEquals_SINT
VAR_INPUT
    Expected : SINT; // SINT expected value
    Actual : SINT; // SINT actual value
    Message : Tc2_System.T_MaxString; // The identifying message for the assertion error
END_VAR
VAR
    TestInstancePath : Tc2_System.T_MaxString;
    AlreadyReported : BOOL;
END_VAR
IF GVL_TcUnit.IgnoreCurrentTest OR GVL_TcUnit.CurrentTestIsFinished THEN
    RETURN;
END_IF

TestInstancePath := AddTestNameToInstancePath(TestInstancePath := FindTestSuiteInstancePath());

AssertResults.ReportResult(ExpectedSize := SIZEOF(Expected),
                           ExpectedTypeClass := IBaseLibrary.TypeClass.TYPE_SINT,
                           ExpectedValue := ADR(Expected),
                           ActualSize := SIZEOF(Actual),
                           ActualTypeClass := IBaseLibrary.TypeClass.TYPE_SINT,
                           ActualValue := ADR(Actual),
                           Message := Message,
                           TestInstancePath := TestInstancePath,
                           AlreadyReported => AlreadyReported);

IF NOT AlreadyReported AND Expected <> Actual THEN
    SetTestFailed(AssertionType := E_AssertionType.Type_SINT,
                  AssertionMessage := Message);

    AssertMessageFormatter.LogAssertFailure(Expected := SINT_TO_STRING(Expected),
                                            Actual := SINT_TO_STRING(Actual),
                                            Message := Message,
                                            TestInstancePath := TestInstancePath);
END_IF
END_METHOD

(*
    Asserts that two STRINGs are equal. If they are not, an assertion error is created.
*)
METHOD PUBLIC AssertEquals_STRING
VAR_INPUT
    Expected : Tc2_System.T_MaxString; // STRING expected value
    Actual : Tc2_System.T_MaxString; // STRING actual value
    Message : Tc2_System.T_MaxString; // The identifying message for the assertion error
END_VAR
VAR
    TestInstancePath : Tc2_System.T_MaxString;
    AlreadyReported : BOOL;
END_VAR
IF GVL_TcUnit.IgnoreCurrentTest OR GVL_TcUnit.CurrentTestIsFinished THEN
    RETURN;
END_IF

TestInstancePath := AddTestNameToInstancePath(TestInstancePath := FindTestSuiteInstancePath());

AssertResults.ReportResult(ExpectedSize := SIZEOF(Expected),
                           ExpectedTypeClass := IBaseLibrary.TypeClass.TYPE_STRING,
                           ExpectedValue := ADR(Expected),
                           ActualSize := SIZEOF(Actual),
                           ActualTypeClass := IBaseLibrary.TypeClass.TYPE_STRING,
                           ActualValue := ADR(Actual),
                           Message := Message,
                           TestInstancePath := TestInstancePath,
                           AlreadyReported => AlreadyReported);

IF NOT AlreadyReported AND (Tc2_Standard.LEN(STR := Expected) <> Tc2_Standard.LEN(STR := Actual) OR (Expected <> Actual)) THEN
    SetTestFailed(AssertionType := E_AssertionType.Type_STRING,
                  AssertionMessage := Message);

    AssertMessageFormatter.LogAssertFailure(Expected := Expected,
                                            Actual := Actual,
                                            Message := Message,
                                            TestInstancePath := TestInstancePath);
END_IF
END_METHOD

(*
    Asserts that two TIMEs are equal. If they are not, an assertion error is created.
*)
METHOD PUBLIC AssertEquals_TIME
VAR_INPUT
    Expected : TIME; // TIME expected value
    Actual : TIME; // TIME actual value
    Message : Tc2_System.T_MaxString; // The identifying message for the assertion error
END_VAR
VAR
    TestInstancePath : Tc2_System.T_MaxString;
    AlreadyReported : BOOL;
END_VAR
IF GVL_TcUnit.IgnoreCurrentTest OR GVL_TcUnit.CurrentTestIsFinished THEN
    RETURN;
END_IF

TestInstancePath := AddTestNameToInstancePath(TestInstancePath := FindTestSuiteInstancePath());

AssertResults.ReportResult(ExpectedSize := SIZEOF(Expected),
                           ExpectedTypeClass := IBaseLibrary.TypeClass.TYPE_TIME,
                           ExpectedValue := ADR(Expected),
                           ActualSize := SIZEOF(Actual),
                           ActualTypeClass := IBaseLibrary.TypeClass.TYPE_TIME,
                           ActualValue := ADR(Actual),
                           Message := Message,
                           TestInstancePath := TestInstancePath,
                           AlreadyReported => AlreadyReported);

IF NOT AlreadyReported AND Expected <> Actual THEN
    SetTestFailed(AssertionType := E_AssertionType.Type_TIME,
                  AssertionMessage := Message);

    AssertMessageFormatter.LogAssertFailure(Expected := TIME_TO_STRING(Expected),
                                            Actual := TIME_TO_STRING(Actual),
                                            Message := Message,
                                            TestInstancePath := TestInstancePath);
END_IF
END_METHOD

(*
    Asserts that two TIME_OF_DAYs are equal. If they are not, an assertion error is created.
*)
METHOD PUBLIC AssertEquals_TIME_OF_DAY
VAR_INPUT
    Expected : TIME_OF_DAY; // TIME_OF_DAY expected value
    Actual : TIME_OF_DAY; // TIME_OF_DAY actual value
    Message : Tc2_System.T_MaxString; // The identifying message for the assertion error
END_VAR
VAR
    TestInstancePath : Tc2_System.T_MaxString;
    AlreadyReported : BOOL;
END_VAR
IF GVL_TcUnit.IgnoreCurrentTest OR GVL_TcUnit.CurrentTestIsFinished THEN
    RETURN;
END_IF

TestInstancePath := AddTestNameToInstancePath(TestInstancePath := FindTestSuiteInstancePath());

AssertResults.ReportResult(ExpectedSize := SIZEOF(Expected),
                           ExpectedTypeClass := IBaseLibrary.TypeClass.TYPE_TIMEOFDAY,
                           ExpectedValue := ADR(Expected),
                           ActualSize := SIZEOF(Actual),
                           ActualTypeClass := IBaseLibrary.TypeClass.TYPE_TIMEOFDAY,
                           ActualValue := ADR(Actual),
                           Message := Message,
                           TestInstancePath := TestInstancePath,
                           AlreadyReported => AlreadyReported);

IF NOT AlreadyReported AND Expected <> Actual THEN
    SetTestFailed(AssertionType := E_AssertionType.Type_TIME_OF_DAY,
                  AssertionMessage := Message);

    AssertMessageFormatter.LogAssertFailure(Expected := TOD_TO_STRING(Expected),
                                            Actual := TOD_TO_STRING(Actual),
                                            Message := Message,
                                            TestInstancePath := TestInstancePath);
END_IF
END_METHOD

(*
    Asserts that two UDINTs are equal. If they are not, an assertion error is created.
*)
METHOD PUBLIC AssertEquals_UDINT
VAR_INPUT
    Expected : UDINT; // UDINT expected value
    Actual : UDINT; // UDINT actual value
    Message : Tc2_System.T_MaxString; // The identifying message for the assertion error
END_VAR
VAR
    TestInstancePath : Tc2_System.T_MaxString;
    AlreadyReported : BOOL;
END_VAR
IF GVL_TcUnit.IgnoreCurrentTest OR GVL_TcUnit.CurrentTestIsFinished THEN
    RETURN;
END_IF

TestInstancePath := AddTestNameToInstancePath(TestInstancePath := FindTestSuiteInstancePath());

AssertResults.ReportResult(ExpectedSize := SIZEOF(Expected),
                           ExpectedTypeClass := IBaseLibrary.TypeClass.TYPE_UDINT,
                           ExpectedValue := ADR(Expected),
                           ActualSize := SIZEOF(Actual),
                           ActualTypeClass := IBaseLibrary.TypeClass.TYPE_UDINT,
                           ActualValue := ADR(Actual),
                           Message := Message,
                           TestInstancePath := TestInstancePath,
                           AlreadyReported => AlreadyReported);

IF NOT AlreadyReported AND Expected <> Actual THEN
    SetTestFailed(AssertionType := E_AssertionType.Type_UDINT,
                  AssertionMessage := Message);

    AssertMessageFormatter.LogAssertFailure(Expected := UDINT_TO_STRING(Expected),
                                            Actual := UDINT_TO_STRING(Actual),
                                            Message := Message,
                                            TestInstancePath := TestInstancePath);
END_IF
END_METHOD

(*
    Asserts that two UINTs are equal. If they are not, an assertion error is created.
*)
METHOD PUBLIC AssertEquals_UINT
VAR_INPUT
    Expected : UINT; // UINT expected value
    Actual : UINT; // UINT actual value
    Message : Tc2_System.T_MaxString; // The identifying message for the assertion error
END_VAR
VAR
    TestInstancePath : Tc2_System.T_MaxString;
    AlreadyReported : BOOL;
END_VAR
IF GVL_TcUnit.IgnoreCurrentTest OR GVL_TcUnit.CurrentTestIsFinished THEN
    RETURN;
END_IF

TestInstancePath := AddTestNameToInstancePath(TestInstancePath := FindTestSuiteInstancePath());

AssertResults.ReportResult(ExpectedSize := SIZEOF(Expected),
                           ExpectedTypeClass := IBaseLibrary.TypeClass.TYPE_UINT,
                           ExpectedValue := ADR(Expected),
                           ActualSize := SIZEOF(Actual),
                           ActualTypeClass := IBaseLibrary.TypeClass.TYPE_UINT,
                           ActualValue := ADR(Actual),
                           Message := Message,
                           TestInstancePath := TestInstancePath,
                           AlreadyReported => AlreadyReported);

IF NOT AlreadyReported AND Expected <> Actual THEN
    SetTestFailed(AssertionType := E_AssertionType.Type_UINT,
                  AssertionMessage := Message);

    AssertMessageFormatter.LogAssertFailure(Expected := UINT_TO_STRING(Expected),
                                            Actual := UINT_TO_STRING(Actual),
                                            Message := Message,
                                            TestInstancePath := TestInstancePath);
END_IF
END_METHOD

(*
    Asserts that two ULINTs are equal. If they are not, an assertion error is created.
*)
METHOD PUBLIC AssertEquals_ULINT
VAR_INPUT
    Expected : ULINT; // ULINT expected value
    Actual : ULINT; // ULINT actual value
    Message : Tc2_System.T_MaxString; // The identifying message for the assertion error
END_VAR
VAR
    TestInstancePath : Tc2_System.T_MaxString;
    AlreadyReported : BOOL;
END_VAR
IF GVL_TcUnit.IgnoreCurrentTest OR GVL_TcUnit.CurrentTestIsFinished THEN
    RETURN;
END_IF

TestInstancePath := AddTestNameToInstancePath(TestInstancePath := FindTestSuiteInstancePath());

AssertResults.ReportResult(ExpectedSize := SIZEOF(Expected),
                           ExpectedTypeClass := IBaseLibrary.TypeClass.TYPE_ULINT,
                           ExpectedValue := ADR(Expected),
                           ActualSize := SIZEOF(Actual),
                           ActualTypeClass := IBaseLibrary.TypeClass.TYPE_ULINT,
                           ActualValue := ADR(Actual),
                           Message := Message,
                           TestInstancePath := TestInstancePath,
                           AlreadyReported => AlreadyReported);

IF NOT AlreadyReported AND Expected <> Actual THEN
    SetTestFailed(AssertionType := E_AssertionType.Type_ULINT,
                  AssertionMessage := Message);

    AssertMessageFormatter.LogAssertFailure(Expected := ULINT_TO_STRING(Expected),
                                            Actual := ULINT_TO_STRING(Actual),
                                            Message := Message,
                                            TestInstancePath := TestInstancePath);
END_IF
END_METHOD

(*
    Asserts that two USINTs are equal. If they are not, an assertion error is created.
*)
METHOD PUBLIC AssertEquals_USINT
VAR_INPUT
    Expected : USINT; // USINT expected value
    Actual : USINT; // USINT actual value
    Message : Tc2_System.T_MaxString; // The identifying message for the assertion error
END_VAR
VAR
    AlreadyReported : BOOL;
    TestInstancePath : Tc2_System.T_MaxString;
END_VAR
IF GVL_TcUnit.IgnoreCurrentTest OR GVL_TcUnit.CurrentTestIsFinished THEN
    RETURN;
END_IF

TestInstancePath := AddTestNameToInstancePath(TestInstancePath := FindTestSuiteInstancePath());

AssertResults.ReportResult(ExpectedSize := SIZEOF(Expected),
                           ExpectedTypeClass := IBaseLibrary.TypeClass.TYPE_USINT,
                           ExpectedValue := ADR(Expected),
                           ActualSize := SIZEOF(Actual),
                           ActualTypeClass := IBaseLibrary.TypeClass.TYPE_USINT,
                           ActualValue := ADR(Actual),
                           Message := Message,
                           TestInstancePath := TestInstancePath,
                           AlreadyReported => AlreadyReported);

IF NOT AlreadyReported AND Expected <> Actual THEN
    SetTestFailed(AssertionType := E_AssertionType.Type_USINT,
                  AssertionMessage := Message);

    AssertMessageFormatter.LogAssertFailure(Expected := USINT_TO_STRING(Expected),
                                            Actual := USINT_TO_STRING(Actual),
                                            Message := Message,
                                            TestInstancePath := TestInstancePath);
END_IF
END_METHOD

(*
    Asserts that two WORDs are equal. If they are not, an assertion error is created.
*)
METHOD PUBLIC AssertEquals_WORD
VAR_INPUT
    Expected : WORD; // WORD expected value
    Actual : WORD; // WORD actual value
    Message : Tc2_System.T_MaxString; // The identifying message for the assertion error
END_VAR
VAR
    TestInstancePath : Tc2_System.T_MaxString;
    AlreadyReported : BOOL;
END_VAR
IF GVL_TcUnit.IgnoreCurrentTest OR GVL_TcUnit.CurrentTestIsFinished THEN
    RETURN;
END_IF

TestInstancePath := AddTestNameToInstancePath(TestInstancePath := FindTestSuiteInstancePath());

AssertResults.ReportResult(ExpectedSize := SIZEOF(Expected),
                           ExpectedTypeClass := IBaseLibrary.TypeClass.TYPE_WORD,
                           ExpectedValue := ADR(Expected),
                           ActualSize := SIZEOF(Actual),
                           ActualTypeClass := IBaseLibrary.TypeClass.TYPE_WORD,
                           ActualValue := ADR(Actual),
                           Message := Message,
                           TestInstancePath := TestInstancePath,
                           AlreadyReported => AlreadyReported);

IF NOT AlreadyReported AND Expected <> Actual THEN
    SetTestFailed(AssertionType := E_AssertionType.Type_WORD,
                  AssertionMessage := Message);

    AssertMessageFormatter.LogAssertFailure(Expected := Tc2_Standard.CONCAT(
                                                            STR1 := '0x',
                                                            STR2 := Tc2_Utilities.WORD_TO_HEXSTR(in := Expected,
                                                                                                 iPrecision := 4,
                                                                                                 bLoCase := FALSE)),
                                            Actual := Tc2_Standard.CONCAT(
                                                            STR1 := '0x',
                                                            STR2 := Tc2_Utilities.WORD_TO_HEXSTR(in := Actual,
                                                                                                 iPrecision := 4,
                                                                                                 bLoCase := FALSE)),
                                            Message := Message,
                                            TestInstancePath := TestInstancePath);
END_IF
END_METHOD

(*
    Asserts that two WSTRINGs are equal. If they are not, an assertion error is created.
*)
METHOD PUBLIC AssertEquals_WSTRING
VAR_INPUT
    Expected : WSTRING(255); // WSTRING expected value
    Actual : WSTRING(255); // WSTRING actual value
    Message : Tc2_System.T_MaxString; // The identifying message for the assertion error
END_VAR
VAR
    TestInstancePath : Tc2_System.T_MaxString;
    AlreadyReported : BOOL;
END_VAR
IF GVL_TcUnit.IgnoreCurrentTest OR GVL_TcUnit.CurrentTestIsFinished THEN
    RETURN;
END_IF

TestInstancePath := AddTestNameToInstancePath(TestInstancePath := FindTestSuiteInstancePath());

AssertResults.ReportResult(ExpectedSize := SIZEOF(Expected),
                           ExpectedTypeClass := IBaseLibrary.TypeClass.TYPE_WSTRING,
                           ExpectedValue := ADR(Expected),
                           ActualSize := SIZEOF(Actual),
                           ActualTypeClass := IBaseLibrary.TypeClass.TYPE_WSTRING,
                           ActualValue := ADR(Actual),
                           Message := Message,
                           TestInstancePath := TestInstancePath,
                           AlreadyReported => AlreadyReported);

IF NOT AlreadyReported AND (Tc2_Standard.WLEN(STR := Expected) <> Tc2_Standard.WLEN(STR := Actual) OR (Expected <> Actual)) THEN
    SetTestFailed(AssertionType := E_AssertionType.Type_WSTRING,
                  AssertionMessage := Message);

    AssertMessageFormatter.LogAssertFailure(Expected := 'Not possible to print EXP unicode WSTRING value',
                                            Actual := 'Not possible to print ACT unicode WSTRING value',
                                            Message := Message,
                                            TestInstancePath := TestInstancePath);
END_IF
END_METHOD

(*
    Asserts that a condition is false. If it is not, an assertion error is created.
*)
METHOD PUBLIC AssertFalse
VAR_INPUT
    Condition : BOOL; // Condition to be checked
    Message : Tc2_System.T_MaxString; // The identifying message for the assertion error
END_VAR
AssertEquals_BOOL(Expected := FALSE, Actual := Condition, Message := Message);
END_METHOD

(*
    Asserts that a condition is true. If it is not, an assertion error is created.
*)
METHOD PUBLIC AssertTrue
VAR_INPUT
    Condition : BOOL; // Condition to be checked
    Message : Tc2_System.T_MaxString; // The identifying message for the assertion error
END_VAR
AssertEquals_BOOL(Expected := TRUE, Actual := Condition, Message := Message);
END_METHOD

METHOD INTERNAL CalculateAndSetNumberOfAssertsForTest
VAR_INPUT
    TestName : Tc2_System.T_MaxString;
END_VAR
VAR
    TestInstancePath : Tc2_System.T_MaxString;
    TotalNumberOfAsserts : UINT;
    NumberOfAsserts : UINT;
    NumberOfArrayAsserts : UINT;
    
    IteratorCounter : UINT;
END_VAR
TestInstancePath := AddTestNameToInstancePath(FindTestSuiteInstancePath());
NumberOfAsserts := AssertResults.GetNumberOfAssertsForTest(CompleteTestInstancePath := TestInstancePath);
NumberOfArrayAsserts := AssertArrayResults.GetNumberOfArrayAssertsForTest(CompleteTestInstancePath := TestInstancePath);
TotalNumberOfAsserts := NumberOfAsserts + NumberOfArrayAsserts;

IF TotalNumberOfAsserts > 0 THEN
    IF NumberOfTests > 0 THEN
        FOR IteratorCounter := 1 TO NumberOfTests BY 1 DO
            IF Tests[IteratorCounter].GetName() = TestName THEN
                Tests[IteratorCounter].SetNumberOfAssertions(NoOfAssertions := TotalNumberOfAsserts);
                RETURN;
            END_IF
        END_FOR
    END_IF
END_IF
END_METHOD

METHOD FB_init : BOOL
VAR_INPUT
    bInitRetains : BOOL; // if TRUE, the retain variables are initialized (warm start / cold start)
    bInCopyCode : BOOL;  // if TRUE, the instance afterwards gets moved into the copy code (online change)
END_VAR
GVL_TcUnit.NumberOfInitializedTestSuites := GVL_TcUnit.NumberOfInitializedTestSuites + 1;    
GVL_TcUnit.TestSuiteAddresses[GVL_TcUnit.NumberOfInitializedTestSuites] := THIS;
END_METHOD

(* Searches for the instance path of the calling function block *)
METHOD PRIVATE FindTestSuiteInstancePath : Tc2_System.T_MaxString
FindTestSuiteInstancePath := GetInstancePath();
END_METHOD

METHOD INTERNAL GetHasStartedRunning : BOOL
GetHasStartedRunning := HasStartedRunning;
END_METHOD

METHOD INTERNAL GetInstancePath : Tc2_System.T_MaxString
GetInstancePath := InstancePath;
END_METHOD

METHOD INTERNAL GetNumberOfFailedTests : UINT
VAR
    Counter : UINT;
    FailedTestsCount : UINT;
    NumberOfTestsToAnalyse : UINT(1..GVL_Param_TcUnit.MaxNumberOfTestSuites);
    NumberOfTestOverArrayLimit : UINT;
END_VAR
(* Limit the test analyse to the max array limit of 'Tests[]' *)
NumberOfTestsToAnalyse := GetNumberOfTestsToAnalyse();
IF GetNumberOfTests() > NumberOfTestsToAnalyse THEN
    NumberOfTestOverArrayLimit := GetNumberOfTests()-NumberOfTestsToAnalyse;
END_IF

FOR Counter := 1 TO NumberOfTestsToAnalyse BY 1 DO
    IF Tests[Counter].IsFailed() THEN
        FailedTestsCount := FailedTestsCount + 1;
    END_IF
END_FOR

GetNumberOfFailedTests := FailedTestsCount + NumberOfTestOverArrayLimit;
END_METHOD

METHOD INTERNAL GetNumberOfSkippedTests : UINT
VAR
    Counter : UINT;
    SkippedTestsCount : UINT;
    NumberOfTestsToAnalyse : UINT(1..GVL_Param_TcUnit.MaxNumberOfTestSuites);
END_VAR
(* Limit the test analyse to the max array limit of 'Tests[]' *)
NumberOfTestsToAnalyse := GetNumberOfTestsToAnalyse();

FOR Counter := 1 TO NumberOfTestsToAnalyse BY 1 DO
    IF Tests[Counter].IsSkipped() THEN
        SkippedTestsCount := SkippedTestsCount + 1;
    END_IF
END_FOR

GetNumberOfSkippedTests := SkippedTestsCount;
END_METHOD

METHOD INTERNAL GetNumberOfSuccessfulTests : UINT
GetNumberOfSuccessfulTests := GetNumberOfTests() - GetNumberOfFailedTests() - GetNumberOfSkippedTests();
END_METHOD

METHOD INTERNAL GetNumberOfTests : UINT
GetNumberOfTests := NumberOfTests;
END_METHOD

METHOD INTERNAL GetNumberOfTestsToAnalyse : UINT
GetNumberOfTestsToAnalyse := MIN(GetNumberOfTests(), GVL_Param_TcUnit.MaxNumberOfTestsForEachTestSuite);
END_METHOD

(* This method returns the test at the n'th position, ranging from 1.. NumberOfTests *)
METHOD INTERNAL GetTestByPosition : FB_Test
VAR_INPUT
    Position : UINT(1..GVL_Param_TcUnit.MaxNumberOfTestsForEachTestSuite);
END_VAR
GetTestByPosition := Tests[Position];
END_METHOD

METHOD INTERNAL GetTestOrderNumber : UINT(0..GVL_Param_TcUnit.MaxNumberOfTestsForEachTestSuite);
VAR_INPUT
    TestName : Tc2_System.T_MaxString;
END_VAR
VAR
    IteratorCounter : UINT;
    NumberOfTestsToAnalyse : UINT(1..GVL_Param_TcUnit.MaxNumberOfTestSuites);
END_VAR
(* Limit the test analyse to the max array limit of 'Tests[]' *)
NumberOfTestsToAnalyse := GetNumberOfTestsToAnalyse();

FOR IteratorCounter := 1 TO NumberOfTestsToAnalyse BY 1 DO
    IF Tests[IteratorCounter].GetName() = TestName THEN
        GetTestOrderNumber := Tests[IteratorCounter].GetTestOrder();
        RETURN;
    END_IF
END_FOR
END_METHOD

METHOD INTERNAL IsTestFinished : BOOL
VAR_INPUT
    TestName : Tc2_System.T_MaxString;
END_VAR
VAR
    IteratorCounter : UINT;
    NumberOfTestsToAnalyse : UINT(0..GVL_Param_TcUnit.MaxNumberOfTestsForEachTestSuite);
END_VAR
(* Limit the test analyse to the max array limit of 'Tests[]' *)
NumberOfTestsToAnalyse := GetNumberOfTestsToAnalyse();

IsTestFinished := FALSE;
FOR IteratorCounter := 1 TO NumberOfTestsToAnalyse BY 1 DO
    IF Tests[IteratorCounter].GetName() = TestName THEN
        IsTestFinished := Tests[IteratorCounter].IsFinished();
        RETURN;
    END_IF
END_FOR
END_METHOD

METHOD ResetTestSuite
VAR
    Counter 				: UINT;
    NumberOfTestsToAnalyse	: UINT(1..GVL_Param_TcUnit.MaxNumberOfTestsForEachTestSuite);
END_VAR
HasStartedRunning := FALSE;

(* Limit the reset to the max array limit of 'Tests[]' *)
NumberOfTestsToAnalyse := MIN(NumberOfTests, GVL_Param_TcUnit.MaxNumberOfTestsForEachTestSuite);

FOR Counter := 1 TO NumberOfTestsToAnalyse BY 1 DO
	(* A test is considered finished if it is finished running (i.e. set by TEST_FINISHED) or if it is skipped/disabled *)
	Tests[Counter].ResetTest();
END_FOR
END_METHOD

METHOD INTERNAL SetHasStartedRunning
HasStartedRunning := TRUE;
END_METHOD

METHOD PRIVATE SetTestFailed
VAR_INPUT
    AssertionType : E_AssertionType;
    AssertionMessage : Tc2_System.T_MaxString;
END_VAR
VAR
    IteratorCounter : UINT;
    NumberOfTestsToAnalyse : UINT(0..GVL_Param_TcUnit.MaxNumberOfTestsForEachTestSuite);
END_VAR
(* Limit the test analyse to the max array limit of 'Tests[]' *)
NumberOfTestsToAnalyse := GetNumberOfTestsToAnalyse();

FOR IteratorCounter := 1 TO NumberOfTestsToAnalyse BY 1 DO
    IF Tests[IteratorCounter].GetName() = GVL_TcUnit.CurrentTestNameBeingCalled THEN
        Tests[IteratorCounter].SetFailed();
        Tests[IteratorCounter].SetAssertionType(AssertType := AssertionType);
        Tests[IteratorCounter].SetAssertionMessage(AssertMessage := AssertionMessage);
    END_IF
END_FOR
END_METHOD

(* Marks the test as finished in this testsuite.
   Returns TRUE if test was found, and FALSE if a test with this name was not found in this testsuite
*)
METHOD INTERNAL SetTestFinished : BOOL;
VAR_INPUT
    TestName : Tc2_System.T_MaxString;
END_VAR
VAR
    IteratorCounter : UINT;
    NumberOfTestsToAnalyse : UINT(0..GVL_Param_TcUnit.MaxNumberOfTestsForEachTestSuite);
END_VAR
(* Limit the test analyse to the max array limit of 'Tests[]' *)
NumberOfTestsToAnalyse := GetNumberOfTestsToAnalyse();
FOR IteratorCounter := 1 TO NumberOfTestsToAnalyse BY 1 DO
    IF Tests[IteratorCounter].GetName() = TestName THEN
        Tests[IteratorCounter].SetFinished();
        SetTestFinished := TRUE;
        RETURN;
    END_IF
END_FOR
SetTestFinished := FALSE;
END_METHOD

END_FUNCTION_BLOCK

(* stored: Version 1.1.0.1, ProductVersion 3.1.4024.11
   POU FB_TestSuite: Id {f80c23f2-119d-406b-ae11-06d1991bf64d}, SpecialFunc None
   Method AddTest: Id {d383011f-6bea-4b05-9018-ea4782ad2837}
   Method AddTestNameToInstancePath: Id {abecfe2f-b0e2-4118-a1c6-bb248556b776}
   Method AreAllTestsFinished: Id {2b211901-49a8-4e51-90e1-4b1e298f9e0c}
   Method AssertArray2dEquals_LREAL: Id {964c2fec-9de7-47ae-bee4-23c559ae4a3f}
   Method AssertArray2dEquals_REAL: Id {dc3b5666-7b5a-49ae-9837-cbb9bedd911a}
   Method AssertArray3dEquals_LREAL: Id {251da4d5-4df8-4eed-b154-a479323eb0d5}
   Method AssertArray3dEquals_REAL: Id {0dc8fccf-4b9a-4206-8d9f-212f576edb04}
   Method AssertArrayEquals_BOOL: Id {3d4059ab-c241-4859-9a9f-090cab6db606}
   Method AssertArrayEquals_BYTE: Id {375a5287-a3e9-4833-ac17-bab8f3f0fdc9}
   Method AssertArrayEquals_DINT: Id {4f0d9b20-0c78-467d-a52a-6badbd5d37cc}
   Method AssertArrayEquals_DWORD: Id {eec9d02d-95a1-4885-9906-ad4b2d0f4cab}
   Method AssertArrayEquals_INT: Id {d54cf111-a7e7-4f51-bdf4-9853e055f62d}
   Method AssertArrayEquals_LINT: Id {d7e53e6b-caed-4867-9ef5-3ccb7ae16bf8}
   Method AssertArrayEquals_LREAL: Id {fbc23ff0-cdf6-43f2-82cd-e6f3a7903664}
   Method AssertArrayEquals_LWORD: Id {7bc0c786-fccc-46e3-b38f-2013c44bfcb0}
   Method AssertArrayEquals_REAL: Id {c42ec40e-0859-4258-a3b2-11b258dab324}
   Method AssertArrayEquals_SINT: Id {133c577e-0641-4157-b42b-46dbf29f788e}
   Method AssertArrayEquals_UDINT: Id {5f690331-57e2-4ea1-b1d7-ab65b52dc848}
   Method AssertArrayEquals_UINT: Id {358571ac-0a0d-4e71-8097-c7943f718fce}
   Method AssertArrayEquals_ULINT: Id {916529a0-57b3-4947-a5b8-e7b9ff17f35f}
   Method AssertArrayEquals_USINT: Id {b3215098-2f26-48bf-a7e4-ee1a0803a968}
   Method AssertArrayEquals_WORD: Id {16eada18-ce2b-459d-a8d9-277e84766935}
   Method AssertEquals: Id {092092ee-35b6-45cc-a1ac-e428e5d747ba}
   Method AssertEquals_BOOL: Id {0c41b405-ea35-4450-93cc-7c3349bdf754}
   Method AssertEquals_BYTE: Id {c039f3f1-9c41-4f5e-93a3-393ce160979a}
   Method AssertEquals_DATE: Id {1645ab79-f969-41aa-a170-f589a5757e7f}
   Method AssertEquals_DATE_AND_TIME: Id {42befc01-2199-49e2-b7ef-cf909b8890f9}
   Method AssertEquals_DINT: Id {b7177b75-64df-4021-85c6-c366f61f5f89}
   Method AssertEquals_DWORD: Id {3ce6ba77-0ab2-46fc-a7c9-978b376b93be}
   Method AssertEquals_INT: Id {7c61106e-9bcd-4577-a949-ab96d8862e41}
   Method AssertEquals_LINT: Id {9dc34017-cbc7-41a9-83a2-941f39cc7271}
   Method AssertEquals_LREAL: Id {205d107c-0a2d-44f7-b68a-eb06720b6a6b}
   Method AssertEquals_LTIME: Id {05ea6378-c553-40a9-9e6b-8f3736f63098}
   Method AssertEquals_LWORD: Id {08b090fb-911b-49fa-a51a-7f5edfd3dd2c}
   Method AssertEquals_REAL: Id {fba4feaf-27d0-4f8b-9014-3895f7bb9cc7}
   Method AssertEquals_SINT: Id {10052dfe-cfcb-4a5a-aa97-151e272ce217}
   Method AssertEquals_STRING: Id {cad7fed3-5db3-4371-9240-856c3c740489}
   Method AssertEquals_TIME: Id {717a0cdd-16a7-4f45-90f3-f5700dba9369}
   Method AssertEquals_TIME_OF_DAY: Id {d892dd01-3d32-4eb1-9f95-980dff16616c}
   Method AssertEquals_UDINT: Id {9c21e8db-62d7-4e5c-8e00-cd508f4f5abc}
   Method AssertEquals_UINT: Id {86b960b9-ebc0-46af-91ed-94a423f501dc}
   Method AssertEquals_ULINT: Id {6f1e7566-33c3-4f9c-b92d-7828feb26211}
   Method AssertEquals_USINT: Id {7f12117a-f0ab-475b-ba47-c8a5c801a9ac}
   Method AssertEquals_WORD: Id {85132cdb-0553-4070-be9a-976fcddd873d}
   Method AssertEquals_WSTRING: Id {74750f5e-0a5e-499f-bc11-ef38c3a2fafb}
   Method AssertFalse: Id {022665a8-9003-4aaa-8ef4-bd39fe196883}
   Method AssertTrue: Id {c415013c-c271-42ba-83ad-6c2c653d8f2e}
   Method CalculateAndSetNumberOfAssertsForTest: Id {a963cb6a-a176-4774-9e1c-6c7896b6a752}
   Method FB_init: Id {9273f5af-0583-448b-bab6-3359f03f9b91}
   Method FindTestSuiteInstancePath: Id {e69a4510-81a2-4d65-94e4-52c06ac49944}
   Method GetHasStartedRunning: Id {73f869b5-0951-4519-8e1e-dd573837cf2e}
   Method GetInstancePath: Id {178fa338-5ed3-417b-8f4d-e9f120ace4b9}
   Method GetNumberOfFailedTests: Id {12e4522b-e67f-439a-af1d-8713231888aa}
   Method GetNumberOfSkippedTests: Id {51a75168-98fa-4d92-8093-efb431316cf0}
   Method GetNumberOfSuccessfulTests: Id {635213dc-96ca-4be6-9c0d-c0454c29d34d}
   Method GetNumberOfTests: Id {6f67c6d5-c29e-4577-8651-51bd6db3ab63}
   Method GetNumberOfTestsToAnalyse: Id {eab9a959-64bd-4b82-9237-0c256b2aadb6}
   Method GetTestByPosition: Id {3795ba6c-bb70-4d36-8d46-fa6431157992}
   Method GetTestOrderNumber: Id {1a921f29-30c3-4fc7-ae04-d4fc89e986b3}
   Method IsTestFinished: Id {1ef139e2-1210-4139-ba5c-329f8493b09c}
   Method ResetTestSuite: Id {d051da2d-891a-473b-a7da-04d07458e0fd}
   Method SetHasStartedRunning: Id {ec167018-f922-4541-86e8-8b70c1684943}
   Method SetTestFailed: Id {79b1664f-2570-4cef-bd6e-d7307d9a7818}
   Method SetTestFinished: Id {1ec94335-80d7-46d3-a0f0-345f8eda2ea4} *)
